Staubli VAL3: clkValve2.pgx

program clkValve2()
begin
  call toggleValve(2)
end
